VAR_GLOBAL
	i_Analog 	    AT %I* :DINT;
	i_AnalogSquare 	AT %I* :DINT;
	q_Led 		    AT %Q* :BOOL;
END_VAR

(* stored: Version 1.1.0.1, ProductVersion 3.1.4024.12
   GVL GVL: Id {2e109e85-6243-451d-b31e-2f2ecaddcb58} *)
